PROGRAM MAIN
VAR
	x : INT;
END_VAR

x := x + 1;

PrgMqttCom();
//Read_Write_DB();

END_PROGRAM

(* stored: Version 1.1.0.1, ProductVersion 3.1.4022.9
   POU MAIN: Id {f4589ac7-1c5b-4964-bf72-fe6b5b2888ef}, SpecialFunc None *)
